FUNCTION_BLOCK FB_UAwriteMock_Failure IMPLEMENTS I_OPCUA_Write
VAR_INPUT
END_VAR
VAR_OUTPUT
END_VAR
VAR
END_VAR

{warning 'add method implementation '}
METHOD start : BOOL
VAR_INPUT
	Execute	: BOOL;
	ConnectionHdl	: DWORD;
	NodeHdl	: DWORD;
	stNodeAddInfo	: Tc3_PLCopen_OpcUa.ST_UANodeAdditionalInfo;
	pVariable	: PVOID;
	cbData	: UDINT;
	Timeout	: TIME := DEFAULT_ADS_TIMEOUT;
END_VAR
VAR_OUTPUT
	Done	: BOOL;
	Busy	: BOOL;
	Error	: BOOL;
	ErrorID	: DWORD;
END_VAR
IF execute THEN
	Error := TRUE;
END_IF
END_METHOD

END_FUNCTION_BLOCK

(* stored: Version 1.1.0.1, ProductVersion 3.1.4024.9
   POU FB_UAwriteMock_Failure: Id {dd5fe2ba-512b-4b30-973b-0f2d77fac84c}, SpecialFunc None
   Method start: Id {dde4d7e4-8bc2-4844-805d-7436a8fcc762} *)
